PROGRAM analogSignals_ex03_1
VAR
	Frawsensor			: REAL;
	weight				: REAL;
	
	LIN_TRAFO 			: FB_Scale;
END_VAR

LIN_TRAFO(
	fIN:= frawsensor, 
	fIN_min:= 0, 
	fIN_max:= 10, 
	fOUT_min:= 0, 
	fOUT_max:= 500, 
	fOUT=> weight);

END_PROGRAM

(* stored: Version 1.1.0.1
   POU analogSignals_ex03_1: Id {68460e71-0926-4dae-aec1-3e9f2107b839}, SpecialFunc None *)
